ABB RobotStudio station: Colocar_Mesa.rspag

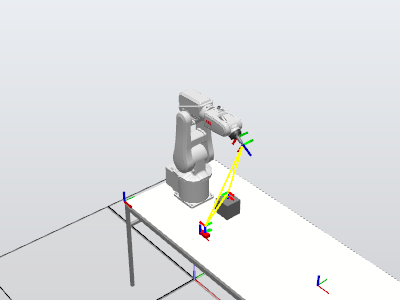
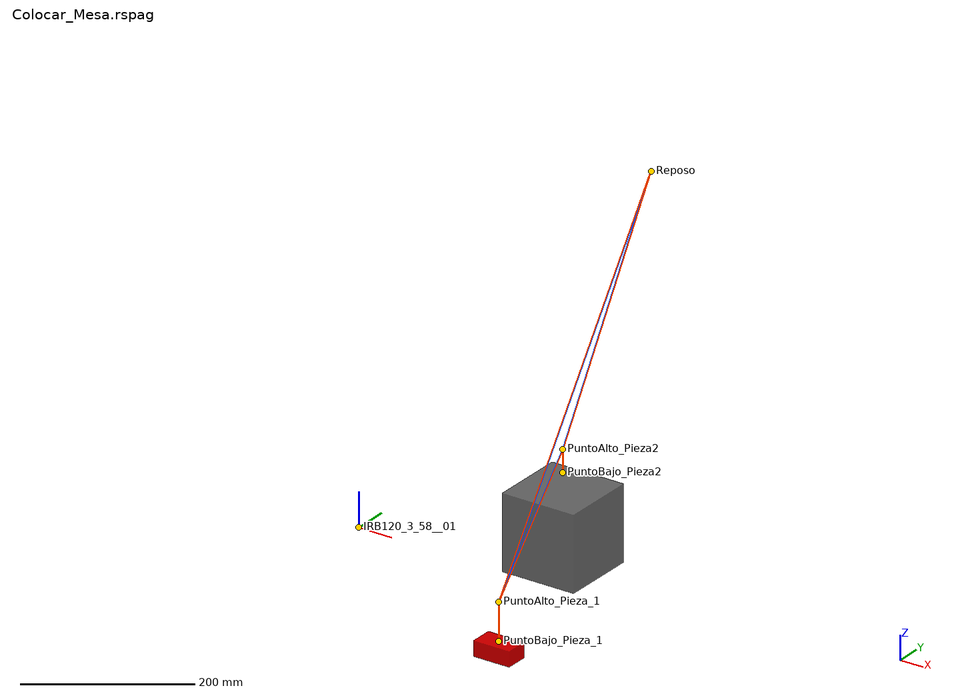
[picture v1: parts stored in the station drawn from their meshes, with robot base, taught points and paths (robot models come from the ABB library and are not in the file)]
--- station ---
Station Práctica2 (saved by RobotStudio 24.3.10885.0)
Controller Controlador2, task T_ROB1: task frame (RAPID world) sits at (1000, 0, 670) mm in the station
Controller Controlador2
  mechanical unit ROB_1: IRB120_3_58__01, 6 joints, base frame (-1000, 0, 0) mm
Layout (positions relative to the parent item):
  - TVentosa [mechanism] at (364.35, 0, 1264) mm, rotated rx 180 ry 60 rz 180 deg
      TCP TVentosa at (0, 0, 51.19) mm
      links: Mi_herramienta
  - LogicGate [smart component, from Components\LogicGate.rslib]
      properties: Operator=NOT; Delay=0
  - LogicGate_2 [smart component, from Components\LogicGate.rslib]
      properties: Operator=AND; Delay=0
  - IRB120_3_58__01 [mechanism, from %ABB.RobotStudio.Models.IRB120%\IRB120_3_58_G_01.rslib] at (0, 0, 670) mm; joint values [0, 0, 0, 0, 0.5236, 0] (rad or m)
  - Table [part, from Práctica2\Table.rslib] at (-220, 350, 670) mm, rotated rx 0 ry 0 rz -90 deg
  - Pieza1 [part] at (325, -185, 690) mm, rotated rx 180 ry 0 rz 180 deg, size 50 x 30 x 20 mm
  - Pieza2 [part], size 100 x 100 x 100 mm
  - CollisionSensor [smart component, from Components\CollisionSensor.rslib]
      properties: Object1=TVentosa; Object2=Pieza1; NearMiss=0.001; Part1=(none); Part2=(none); CollisionType=0
  - Attacher [smart component, from Components\Attacher.rslib]
      properties: Parent=TVentosa; Flange=0; Child=Pieza1; Mount=true; Offset=[0 0 0]; Orientation=[0 0 0]
  - Detacher [smart component, from Components\Detacher.rslib]
      properties: Child=Pieza1; KeepPosition=true
Attachment: TVentosa is attached to IRB120_3_58__01 / Link6
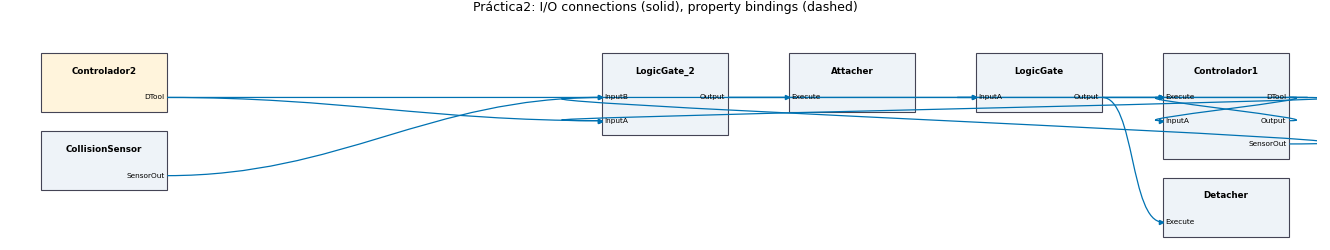
Station logic (signal -> signal, property => property):
  Controlador1.DTool -> Attacher.Execute
  Controlador1.DTool -> LogicGate_2.InputA
  LogicGate_2.Output -> Detacher.Execute
  Controlador1.DTool -> LogicGate.InputA
  LogicGate.Output -> Detacher.Execute
  CollisionSensor.SensorOut -> LogicGate_2.InputB
  Controlador1.DTool -> LogicGate_2.InputA
  LogicGate_2.Output -> Attacher.Execute
  Controlador2.DTool -> LogicGate_2.InputA
  Controlador2.DTool -> LogicGate.InputA
  CollisionSensor.SensorOut -> LogicGate_2.InputB
  LogicGate_2.Output -> Attacher.Execute
  LogicGate.Output -> Detacher.Execute

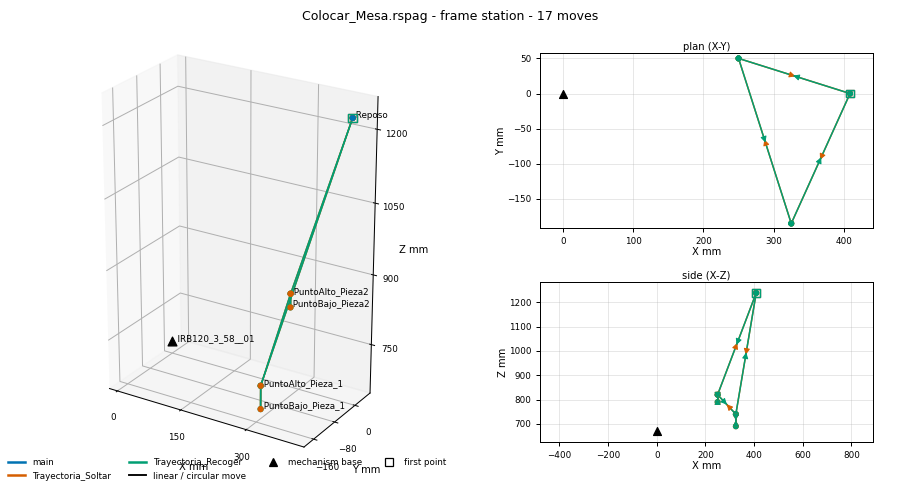
[picture p0: tool path of Colocar_Mesa.rspag in frame station, 17 of 17 moves have a stored position in this frame; points joined in program order, loops and branches not executed]
--- Backups/Controlador2/RAPID/TASK1/PROGMOD/CalibData.mod ---
MODULE CalibData
    PERS tooldata TVentosa:=[TRUE,[[0,0,51.19],[1,0,0,0]],[0.1,[0,0,1],[1,0,0,0],0,0,0]];
    TASK PERS wobjdata WO_Pieza1:=[FALSE,TRUE,"",[[-1220,-350,0],[1,0,0,0]],[[520,150,0],[1,0,0,0]]];
    TASK PERS wobjdata WO_Pieza2:=[FALSE,TRUE,"",[[-1220,-350,0],[1,0,0,0]],[[420,350,0],[1,0,0,0]]];
ENDMODULE

--- Backups/Controlador2/RAPID/TASK1/PROGMOD/Module1.mod ---
MODULE Module1
    CONST robtarget Reposo:=[[-591.315,0,568.405],[0.5,0,0.866025404,0],[0,0,0,0],[9E+09,9E+09,9E+09,9E+09,9E+09,9E+09]];
    CONST robtarget PuntoAlto_Pieza_1:=[[25,15,70],[0,0,1,0],[-1,0,-1,0],[9E+09,9E+09,9E+09,9E+09,9E+09,9E+09]];
    CONST robtarget PuntoBajo_Pieza_1:=[[25,15,20],[0,0,1,0],[0,0,0,0],[9E+09,9E+09,9E+09,9E+09,9E+09,9E+09]];
    CONST robtarget PuntoAlto_Pieza2:=[[50,50,150],[0,1,0,0],[0,0,-2,0],[9E+09,9E+09,9E+09,9E+09,9E+09,9E+09]];
    CONST robtarget PuntoBajo_Pieza2:=[[50,50,120],[0,1,0,0],[0,0,-2,0],[9E+09,9E+09,9E+09,9E+09,9E+09,9E+09]];
    !***********************************************************
    !
    ! Módulo:  Module1
    !
    ! Descripción:
    !   <Introduzca la descripción aquí>
    !
    ! Autor: Maya
    !
    ! Versión: 1.0
    !
    !***********************************************************


    !***********************************************************
    !
    ! Procedimiento Main
    !
    !   Este es el punto de entrada de su programa
    !
    !***********************************************************
    PROC main()
        ! Si la entrada DI0 vale 1, ejecuta las trayectorias
        IF DI0=1 THEN
            Trayectoria_Soltar;
            !LLevar de 1 a 2
            WaitTime 1;
            Trayectoria_Recoger;
            !Llevar de 2 a 1

        ! Si la entrada DI0 vale 0, tras ejecutar las trayectorias, se parará la ejecución y se volverá a la posición de reposo
        ELSE
            MoveL Reposo,v500,fine,TVentosa\WObj:=wobj0;
        ENDIF
    ENDPROC

    PROC Trayectoria_Soltar()
        MoveL Reposo,v500,fine,TVentosa\WObj:=wobj0;
        MoveL PuntoAlto_Pieza_1,v500,fine,TVentosa\WObj:=WO_Pieza1;
        MoveL PuntoBajo_Pieza_1,v500,fine,TVentosa\WObj:=WO_Pieza1;   ! Punto de contacto
        SetDO DTool,1;  ! ACTIVAR VENTOSA
        WaitTime 0.5;  ! Pausa para asegurar el agarre
        MoveL PuntoAlto_Pieza_1,v500,fine,TVentosa\WObj:=WO_Pieza1;
        MoveL PuntoAlto_Pieza2,v500,fine,TVentosa\WObj:=WO_Pieza2;
        MoveL PuntoBajo_Pieza2,v500,fine,TVentosa\WObj:=WO_Pieza2;   ! Llegada al punto de dejada en la pieza 2
        SetDO Dtool,0; ! DESACTIVAR VENTOSA
        MoveL PuntoAlto_Pieza2,v500,fine,TVentosa\WObj:=WO_Pieza2;
        MoveL Reposo,v500,fine,TVentosa\WObj:=wobj0;
    ENDPROC

    PROC Trayectoria_Recoger()
        MoveL Reposo,v500,fine,TVentosa\WObj:=wobj0;
        MoveL PuntoAlto_Pieza2,v500,fine,TVentosa\WObj:=WO_Pieza2;
        MoveL PuntoBajo_Pieza2,v500,fine,TVentosa\WObj:=WO_Pieza2;   ! Punto de contacto
        SetDO DTool,1;   ! ACTIVAR VENTOSA
        WaitTime 0.5;    ! Pausa para asegurar el agarre
        MoveL PuntoAlto_Pieza2,v500,fine,TVentosa\WObj:=WO_Pieza2;
        MoveL PuntoAlto_Pieza_1,v500,fine,TVentosa\WObj:=WO_Pieza1;
        MoveL PuntoBajo_Pieza_1,v500,fine,TVentosa\WObj:=WO_Pieza1;  ! Llegada al punto de dejada en el origen de la pieza 1
        SetDO Dtool,0; ! DESACTIVAR VENTOSA
        MoveL PuntoAlto_Pieza_1,v500,fine,TVentosa\WObj:=WO_Pieza1;
        MoveL Reposo,v500,fine,TVentosa\WObj:=wobj0;
    ENDPROC
ENDMODULE

--- Backups/Controlador2/SYSPAR/EIO.cfg ---
EIO:CFG_1.0:6:1::
#
EIO_SIGNAL:

      -Name "DTool" -SignalType "DO"

      -Name "DI0" -SignalType "DI"
